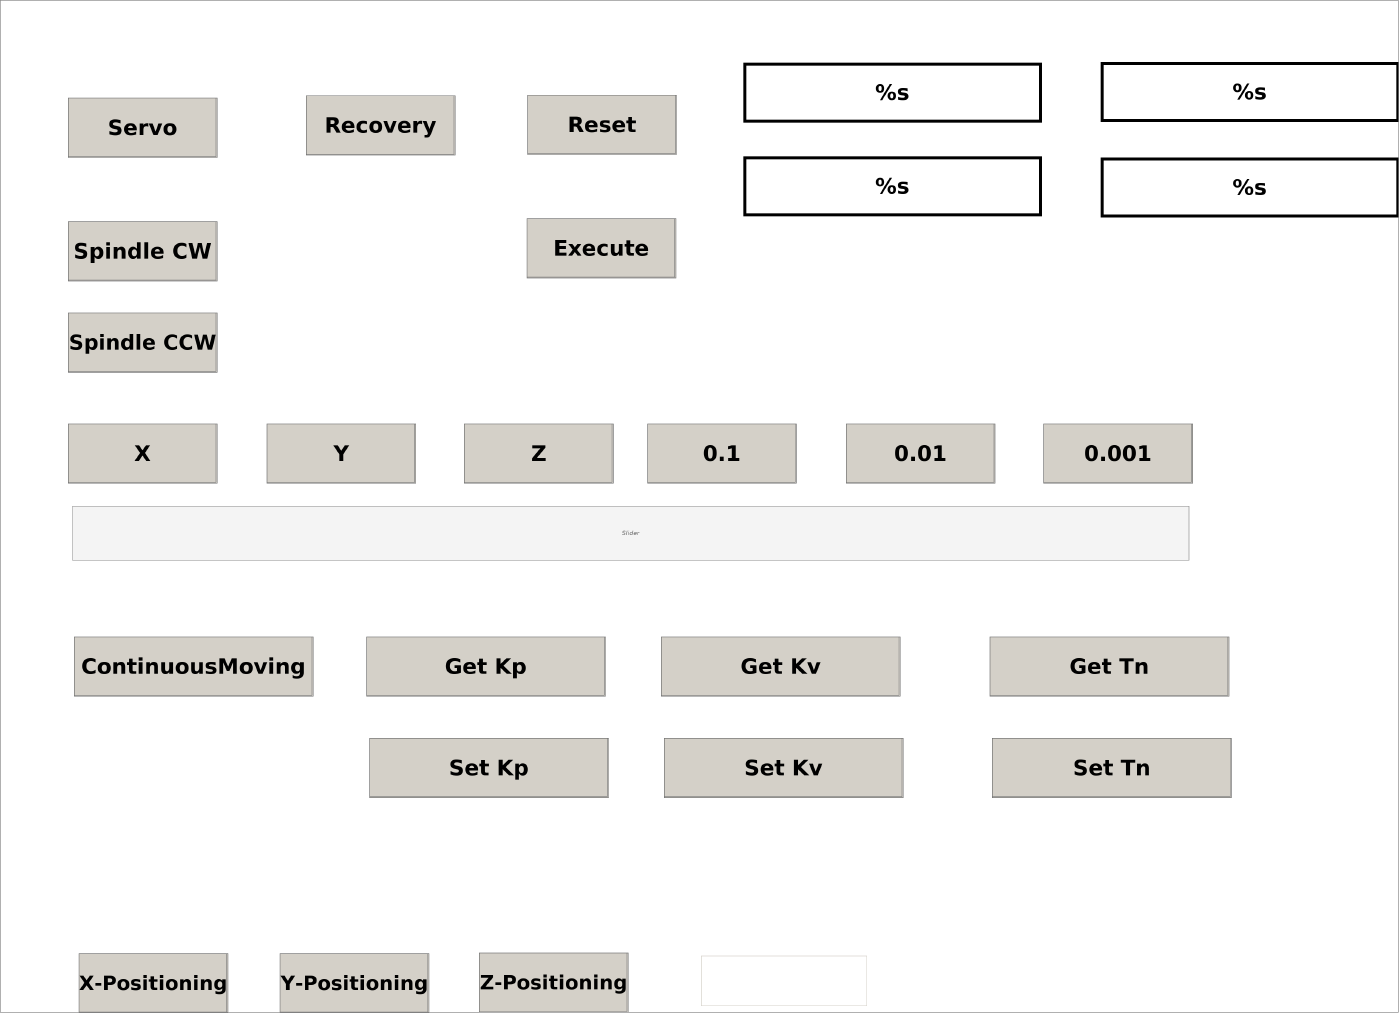
VISUALIZATION TestHMI  // 2345x1698
    Button (114,164 250x100), "Servo", colour toggle: MAIN.MockPanel.ServoOn
        toggle MAIN.MockPanel.ServoOn
    Button (114,371 250x100), "Spindle CW", colour toggle: MAIN.SpindleCW, input disabled if: MAIN.SpindleCCW
        toggle MAIN.SpindleCW
    Button (114,524 250x100), "Spindle CCW", colour toggle: MAIN.SpindleCCW, input disabled if: MAIN.SpindleCW
        toggle MAIN.SpindleCCW
    Slider (121,848 1872x91), variable: MAIN.IncrementalPos, scale -20..20
    Button (114,710 250x100), "X", colour toggle: MAIN.Axis_X
        toggle MAIN.Axis_X
        OnMouseDown: execute { MAIN.MockPanel.Handwheel_EnabledAxisNum := 1; }
    Button (447,710 250x100), "Y", colour toggle: MAIN.Axis_Y
        toggle MAIN.Axis_Y
        OnMouseDown: execute { MAIN.MockPanel.Handwheel_EnabledAxisNum := 2; }
    Button (778,710 250x100), "Z", colour toggle: MAIN.Axis_Z
        toggle MAIN.Axis_Z
        OnMouseDown: execute { MAIN.MockPanel.Handwheel_EnabledAxisNum := 3; }
    Rectangle (1246,105 500x100), "%s", text list: 'AxisGroupStateList', text index: MAIN.AxisGroupStateListId
    Rectangle (1246,262 500x100), "%s", text list: 'SpindleStateList', text index: MAIN.SpindleStateListId
    Button (1085,710 250x100), "0.1", colour toggle: MAIN.Ratio_01
        toggle MAIN.Ratio_01
        OnMouseDown: execute { MAIN.MockPanel.Handwheel_EnabledAxisNum := 1; }
    Button (1418,710 250x100), "0.01", colour toggle: MAIN.Ratio_001
        toggle MAIN.Ratio_001
        OnMouseDown: execute { MAIN.MockPanel.Handwheel_EnabledAxisNum := 2; }
    Button (1749,710 250x100), "0.001", colour toggle: MAIN.Ratio_0001
        toggle MAIN.Ratio_0001
        OnMouseDown: execute { MAIN.MockPanel.Handwheel_EnabledAxisNum := 3; }
    Rectangle (1845,104 500x100), "%s", text list: 'MainStateList', text index: MAIN.MainStateListId
    Rectangle (1845,264 500x100), "%s", text list: 'SafetyStatusList', text index: MAIN.SafetyStatusListId
    Button (513,160 250x100), "Recovery", colour toggle: MAIN.Recovery
        toggle MAIN.Recovery
    Button (884,159 250x100), "Reset", colour toggle: MAIN.MockPanel.Reset
        toggle MAIN.MockPanel.Reset
    Button (124,1067 401x100), "ContinuousMoving", colour toggle: MAIN.ContinuousMoving
        toggle MAIN.ContinuousMoving
        OnMouseDown: execute { MAIN.MockPanel.Handwheel_EnabledAxisNum := 1; }
    Button (614,1067 401x100), "Get Kp", colour toggle: MAIN.GetParamKpValue
        toggle MAIN.GetParamKpValue
        OnMouseDown: execute { MAIN.MockPanel.Handwheel_EnabledAxisNum := 1; }
    Button (619,1237 401x100), "Set Kp", colour toggle: MAIN.SetParamKpValue
        toggle MAIN.SetParamKpValue
        OnMouseDown: execute { MAIN.MockPanel.Handwheel_EnabledAxisNum := 1; }
    Button (1108,1067 401x100), "Get Kv", colour toggle: MAIN.GetParamKvValue
        toggle MAIN.GetParamKvValue
        OnMouseDown: execute { MAIN.MockPanel.Handwheel_EnabledAxisNum := 1; }
    Button (1659,1067 401x100), "Get Tn", colour toggle: MAIN.GetParamTnValue
        toggle MAIN.GetParamTnValue
        OnMouseDown: execute { MAIN.MockPanel.Handwheel_EnabledAxisNum := 1; }
    Button (1663,1237 401x100), "Set Tn", colour toggle: MAIN.SetParamTnValue
        toggle MAIN.SetParamTnValue
        OnMouseDown: execute { MAIN.MockPanel.Handwheel_EnabledAxisNum := 1; }
    Button (1113,1237 401x100), "Set Kv", colour toggle: MAIN.SetParamKvValue
        toggle MAIN.SetParamKvValue
        OnMouseDown: execute { MAIN.MockPanel.Handwheel_EnabledAxisNum := 1; }
    Button (883,366 250x100), "Execute", colour toggle: MAIN.MockPanel.Execute
        toggle MAIN.MockPanel.Execute
    Button (132,1598 250x100), "X-Positioning", colour toggle: MAIN.Position_X
        toggle MAIN.Position_X
        OnMouseDown: execute { MAIN.MockPanel.Handwheel_EnabledAxisNum := 2; }
    Button (803,1597 250x100), "Z-Positioning", colour toggle: MAIN.Position_Z
        toggle MAIN.Position_Z
        OnMouseDown: execute { MAIN.MockPanel.Handwheel_EnabledAxisNum := 2; }
    Button (469,1598 250x100), "Y-Positioning", colour toggle: MAIN.Position_Y
        toggle MAIN.Position_Y
        OnMouseDown: execute { MAIN.MockPanel.Handwheel_EnabledAxisNum := 2; }
    Textfield (1175,1602 278x84)
END_VISUALIZATION

(* stored: Version 1.1.0.1, ProductVersion 3.1.4024.12
   Visu TestHMI: Id {e24fc235-7e11-49f0-8a06-9cbbf9a25ae1} *)
